// TIA Portal V17 export
// export: Created 2024-08-20T10:59:42.8062994Z, ExportSetting WithDefaults, DisplayName Totally Integrated Automation Portal, DisplayVersion V17 Update 4, DisplayName TIA Portal Openness, DisplayVersion V17 Update 4, DisplayName TIA Portal Version Control Interface, DisplayVersion V17, DisplayName STEP 7 Professional, DisplayVersion V17 Update 4, DisplayName STEP 7 Safety, DisplayVersion V17, DisplayName WinCC Advanced, DisplayVersion V17 Update 4
DATA_BLOCK "STATUS"   // DB302
{ S7_Optimized_Access := 'FALSE' }
VERSION : 0.1
// stored: AutoNumber false, DBAccessibleFromOPCUA true, IsOnlyStoredInLoadMemory false, IsWriteProtectedInAS false
   VAR
      "SO-203-06A-YI" : Bool;   // Soprador tanque de aeração intertravado
      "SO-203-06B-YI" : Bool;   // Soprador tanque de aeração intertravado
      "SO-203-06C-YI" : Bool;   // Soprador tanque de aeração intertravado
      "SO-203-06D-YI" : Bool;   // Soprador tanque de aeração intertravado
      "SO-203-06E-YI" : Bool;   // Soprador tanque de aeração intertravado
      "SO-203-06F-YI" : Bool;   // Soprador tanque de aeração intertravado
      "MB-01-YSP" : Bool;   // MB-01 selecionada como principal
      "MB-02-YSP" : Bool;   // MB-02 selecionada como principal
      "MB-04-YSP" : Bool;   // MB-03 selecionada como principal
      "MB-03-YSP" : Bool;   // MB-03 selecionada como principal
      "MB-01-YC1" : Bool;   // MB-01 selecionada como complementar 1
      "MB-02-YC1" : Bool;   // MB-02 selecionada como complementar 1
      "MB-04-YC1" : Bool;   // MB-03 selecionada como complementar 1
      "MB-03-YC1" : Bool;   // MB-03 selecionada como complementar 1
      "MB-01-YC2" : Bool;   // MB-01 selecionada como complementar 2
      "MB-02-YC2" : Bool;   // MB-02 selecionada como complementar 2
      "MB-04-YC2" : Bool;   // MB-03 selecionada como complementar 2
      "MB-03-YC2" : Bool;   // MB-03 selecionada como complementar 2
   END_VAR
BEGIN
END_DATA_BLOCK
